// TwinCAT 3 PLC project PlcCode
// ProgramVersion: 3.1.4024.12
// libraries:
//   Tc2_Standard, * (Beckhoff Automation GmbH)
//   Tc2_System, * (Beckhoff Automation GmbH)
//   Tc2_Utilities, * (Beckhoff Automation GmbH)
//   Tc3_IotBase, * (Beckhoff Automation GmbH)
//   Tc3_JsonXml, * (Beckhoff Automation GmbH)
//   Tc3_Module, * (Beckhoff Automation GmbH)
// project tree:
//   GVLs/ GVL.TcGVL
//   / PlcTask.TcTTO
//   POUs/ MAIN.TcPOU
//   ReadConfigFile/CELLS_INFO_STRUCTURES/Development/ DUT_STRUCT_C000000_DEV.TcDUT (not stored), DUT_STRUCT_C000001_DEV.TcDUT (not stored), DUT_STRUCT_C000002_DEV.TcDUT, DUT_STRUCT_C000003_DEV.TcDUT (not stored), DUT_STRUCT_C000004_DEV.TcDUT (not stored), DUT_STRUCT_C000005_DEV.TcDUT, DUT_STRUCT_C000006_DEV.TcDUT (not stored), DUT_STRUCT_C000007_DEV.TcDUT (not stored), DUT_STRUCT_C000008_DEV.TcDUT, DUT_STRUCT_C000009_DEV.TcDUT (not stored), DUT_STRUCT_C000010_DEV.TcDUT (not stored), DUT_STRUCT_C000012_DEV.TcDUT, DUT_STRUCT_LINECONTROLLER_DEV.TcDUT, DUT_STRUCT_TRACKSERVER_DEV.TcDUT
//   ReadConfigFile/CELLS_INFO_STRUCTURES/Production/ DUT_STRUCT_C000000_PROD.TcDUT, DUT_STRUCT_C000001_PROD.TcDUT (not stored), DUT_STRUCT_C000002_PROD.TcDUT, DUT_STRUCT_C000003_PROD.TcDUT (not stored), DUT_STRUCT_C000004_PROD.TcDUT, DUT_STRUCT_C000005_PROD.TcDUT (not stored), DUT_STRUCT_C000006_PROD.TcDUT, DUT_STRUCT_C000007_PROD.TcDUT (not stored), DUT_STRUCT_C000008_PROD.TcDUT (not stored), DUT_STRUCT_C000009_PROD.TcDUT, DUT_STRUCT_C000010_PROD.TcDUT (not stored), DUT_STRUCT_C000012_PROD.TcDUT (not stored), DUT_STRUCT_LINECONTROLLER_PROD.TcDUT, DUT_STRUCT_TRACKSERVER_PROD.TcDUT
//   ReadConfigFile/ DUT_STRUCT_VARIABLES.TcDUT, FB_HttpGet.TcPOU, FB_ReadFile.TcPOU, ST_ReceivedData.TcDUT (not stored)
// real-time tasks:
//   TASK PlcTask: cycle T#10ms, priority 20, ADS port 350
//   TASK PlcTask1: cycle T#10ms, priority 21, ADS port 351

CONFIGURATION PlcCode
    RESOURCE PLC ON TwinCAT3
        TASK PlcTask(INTERVAL := T#10ms, PRIORITY := 20);
        PROGRAM MAIN WITH PlcTask : MAIN;
    END_RESOURCE
END_CONFIGURATION

// ---- ReadConfigFile/CELLS_INFO_STRUCTURES/Development/DUT_STRUCT_C000002_DEV.TcDUT
TYPE DUT_STRUCT_C000002_DEV :
STRUCT
	sCellName			:STRING := 'C000002';
	sIpAddress			:STRING := '';
	sAmsNetId			:STRING := '';
	sOpcUaURL			:STRING := 'opc.tcp://:4840';
	sStation1			:STRING := 'S000007';
END_STRUCT
END_TYPE

// ---- ReadConfigFile/CELLS_INFO_STRUCTURES/Development/DUT_STRUCT_C000005_DEV.TcDUT
TYPE DUT_STRUCT_C000005_DEV :
STRUCT
	sCellName			:STRING := 'C000005';
	sIpAddress			:STRING := '';
	sAmsNetId			:STRING := '';
	sOpcUaURL			:STRING := 'opc.tcp://:4840';
	sStation1			:STRING := 'S000001';
END_STRUCT
END_TYPE

// ---- ReadConfigFile/CELLS_INFO_STRUCTURES/Development/DUT_STRUCT_C000008_DEV.TcDUT
TYPE DUT_STRUCT_C000008_DEV :
STRUCT
	sCellName			:STRING := 'C000008';
	sIpAddress			:STRING := '';
	sAmsNetId			:STRING := '';
	sOpcUaURL			:STRING := 'opc.tcp://:4840';
	sStation1			:STRING := 'S000005';
END_STRUCT
END_TYPE

// ---- ReadConfigFile/CELLS_INFO_STRUCTURES/Development/DUT_STRUCT_C000012_DEV.TcDUT
TYPE DUT_STRUCT_C000012_DEV :
STRUCT
	sCellName			:STRING := 'C000012';
	sIpAddress			:STRING := '';
	sAmsNetId			:STRING := '';
	sOpcUaURL			:STRING := 'opc.tcp://:4840';
	sStation1			:STRING := 'S000010';
END_STRUCT
END_TYPE

// ---- ReadConfigFile/CELLS_INFO_STRUCTURES/Development/DUT_STRUCT_LINECONTROLLER_DEV.TcDUT
TYPE DUT_STRUCT_LINECONTROLLER_DEV :
STRUCT
	sCellName			:STRING := 'LINECONTROLLER';
	sIpAddress			:STRING := '10.155.180.8';
	sAmsNetId			:STRING := '';
END_STRUCT
END_TYPE

// ---- ReadConfigFile/CELLS_INFO_STRUCTURES/Development/DUT_STRUCT_TRACKSERVER_DEV.TcDUT
TYPE DUT_STRUCT_TRACKSERVER_DEV :
STRUCT
	sCellName			:STRING := 'TRACKSERVER';
	sIpAddress			:STRING := '10.155.180.10';
	sAmsNetId			:STRING := '10.155.180.10.1.1';
END_STRUCT
END_TYPE

// ---- ReadConfigFile/CELLS_INFO_STRUCTURES/Production/DUT_STRUCT_C000000_PROD.TcDUT
TYPE DUT_STRUCT_C000000_PROD :
STRUCT
	sCellName			:STRING := 'C000000';
	sIpAddress			:STRING := '10.38.190.130';
	sAmsNetId			:STRING := '10.38.190.130.1.1';
	sOpcUaURL			:STRING := 'opc.tcp://10.38.190.130:4840';
	sUhfRfidOpcUaURL	:STRING := 'opc.tcp://10.38.190.132:4840';
	sHfRfidOpcUaURL		:STRING := 'opc.tcp://10.38.190.134:4840';
	sStation1			:STRING := 'S00000A';
END_STRUCT
END_TYPE

// ---- ReadConfigFile/CELLS_INFO_STRUCTURES/Production/DUT_STRUCT_C000002_PROD.TcDUT
TYPE DUT_STRUCT_C000002_PROD :
STRUCT
	sCellName			:STRING := 'C000002';
	sIpAddress			:STRING := '10.38.191.20';
	sAmsNetId			:STRING := '10.38.191.20.1.1';
	sOpcUaURL			:STRING := 'opc.tcp://10.38.191.20:4840';
	sStation1			:STRING := 'S000007';
END_STRUCT
END_TYPE

// ---- ReadConfigFile/CELLS_INFO_STRUCTURES/Production/DUT_STRUCT_C000004_PROD.TcDUT
TYPE DUT_STRUCT_C000004_PROD :
STRUCT
	sCellName			:STRING := 'C000004';
	sIpAddress			:STRING := '10.38.190.201';
	sAmsNetId			:STRING := '10.38.190.201.1.1';
	sOpcUaURL			:STRING := 'opc.tcp://10.38.190.201:4840';
	sStation1			:STRING := 'S000003';
END_STRUCT
END_TYPE

// ---- ReadConfigFile/CELLS_INFO_STRUCTURES/Production/DUT_STRUCT_C000006_PROD.TcDUT
TYPE DUT_STRUCT_C000006_PROD :
STRUCT
	sCellName			:STRING := 'C000006';
	sIpAddress			:STRING := '10.38.190.200';
	sAmsNetId			:STRING := '10.38.190.200.1.1';
	sOpcUaURL			:STRING := 'opc.tcp://10.38.190.200:4840';
	sStation1			:STRING := 'S000002';
END_STRUCT
END_TYPE

// ---- ReadConfigFile/CELLS_INFO_STRUCTURES/Production/DUT_STRUCT_C000009_PROD.TcDUT
TYPE DUT_STRUCT_C000009_PROD :
STRUCT
	sCellName			:STRING := 'C000009';
	sIpAddress			:STRING := '10.38.191.60';
	sAmsNetId			:STRING := '10.38.191.60.1.1';
	sOpcUaURL			:STRING := 'opc.tcp://10.38.191.60:4840';
	sUhfRfidOpcUaURL	:STRING := 'opc.tcp://10.38.190.132:4840';
	sHfRfidOpcUaURL		:STRING := 'opc.tcp://10.38.191.66:4840';
	sStation1			:STRING := 'S000004';
	sLastingPC			:STRING := '10.38.191.65';
END_STRUCT
END_TYPE

// ---- ReadConfigFile/CELLS_INFO_STRUCTURES/Production/DUT_STRUCT_LINECONTROLLER_PROD.TcDUT
TYPE DUT_STRUCT_LINECONTROLLER_PROD :
STRUCT
	sCellName			:STRING := 'LINECONTROLLER';
	sIpAddress			:STRING := '10.38.190.120';
	sAmsNetId			:STRING := '';
END_STRUCT
END_TYPE

// ---- ReadConfigFile/CELLS_INFO_STRUCTURES/Production/DUT_STRUCT_TRACKSERVER_PROD.TcDUT
TYPE DUT_STRUCT_TRACKSERVER_PROD :
STRUCT
	sCellName			:STRING := 'TRACKSERVER';
	sIpAddress			:STRING := '10.38.190.121';
	sAmsNetId			:STRING := '10.38.190.121.1.1';
END_STRUCT
END_TYPE

// ---- ReadConfigFile/DUT_STRUCT_VARIABLES.TcDUT
TYPE DUT_STRUCT_VARIABLES :
STRUCT
	sCellName			:STRING;
	sIpAddress			:STRING;
	sAmsNetId			:STRING;
	sOpcUaURL			:STRING;
	sUhfRfidOpcUaURL	:STRING;
	sHfRfidOpcUaURL		:STRING;
	sStation1			:STRING;
	sStation2			:STRING;
END_STRUCT
END_TYPE

// ---- GVLs/GVL.TcGVL
{attribute 'qualified_only'}
VAR_GLOBAL
	
	// vars for JSON & HTTP GET response
	sString						:ARRAY[0..100] OF STRING(255);
	jsonFileResult 				:STRING(501);

	// repo info
	sRelease					:STRING;
	sCommitID					:STRING;
	sTag						:STRING;
	
	// cells info
	C000000						:DUT_STRUCT_VARIABLES;
	C000001						:DUT_STRUCT_VARIABLES;
	C000002						:DUT_STRUCT_VARIABLES;
	C000003						:DUT_STRUCT_VARIABLES;
	C000004						:DUT_STRUCT_VARIABLES;
	C000005						:DUT_STRUCT_VARIABLES;
	C000006						:DUT_STRUCT_VARIABLES;
	C000007						:DUT_STRUCT_VARIABLES;
	C000008						:DUT_STRUCT_VARIABLES;
	C000009						:DUT_STRUCT_VARIABLES;
	C000010						:DUT_STRUCT_VARIABLES;
	C000012						:DUT_STRUCT_VARIABLES;
	LineController				:DUT_STRUCT_VARIABLES;
	Trackserver					:DUT_STRUCT_VARIABLES;
	
	// cells info for PRODUCTION
//	C000000_PROD				:DUT_STRUCT_C000000_PROD;
//	C000001_PROD				:DUT_STRUCT_C000001_PROD;
//	C000002_PROD				:DUT_STRUCT_C000002_PROD;
//	C000003_PROD				:DUT_STRUCT_C000003_PROD;
//	C000004_PROD				:DUT_STRUCT_C000004_PROD;
//	C000005_PROD				:DUT_STRUCT_C000005_PROD;
//	C000006_PROD				:DUT_STRUCT_C000006_PROD;
//	C000007_PROD				:DUT_STRUCT_C000007_PROD;
//	C000008_PROD				:DUT_STRUCT_C000008_PROD;
//	C000009_PROD				:DUT_STRUCT_C000009_PROD;
//	C000010_PROD				:DUT_STRUCT_C000010_PROD;
//	C000012_PROD				:DUT_STRUCT_C000012_PROD;
//	TrackServer_PROD			:DUT_STRUCT_TRACKSERVER_PROD;
//	LineController_PROD			:DUT_STRUCT_LINECONTROLLER_PROD;
	
//	// cells info for DEVELOPMENT
//	C000000_DEV					:DUT_STRUCT_C000000_DEV;
//	C000001_DEV					:DUT_STRUCT_C000001_DEV;
//	C000002_DEV					:DUT_STRUCT_C000002_DEV;
//	C000003_DEV					:DUT_STRUCT_C000003_DEV;
//	C000004_DEV					:DUT_STRUCT_C000004_DEV;
//	C000005_DEV					:DUT_STRUCT_C000005_DEV;
//	C000006_DEV					:DUT_STRUCT_C000006_DEV;
//	C000007_DEV					:DUT_STRUCT_C000007_DEV;
//	C000008_DEV					:DUT_STRUCT_C000008_DEV;
//	C000009_DEV					:DUT_STRUCT_C000009_DEV;
//	C000010_DEV					:DUT_STRUCT_C000010_DEV;
//	C000012_DEV					:DUT_STRUCT_C000012_DEV;
//	TrackServer_DEV				:DUT_STRUCT_TRACKSERVER_DEV;
//	LineController_DEV			:DUT_STRUCT_LINECONTROLLER_DEV;
END_VAR

// ---- POUs/MAIN.TcPOU
PROGRAM MAIN

VAR
	// develop branch
	fbReadFile					:FB_ReadFile;
	bHttpGet					:BOOL := TRUE;

    fbHttpClient				:FB_IotHttpClient := (sHostName:='api.github.com', bKeepAlive:=TRUE, tConnectionTimeout:=T#10S);
    fbHttpGetOpen				:FB_HttpGet;
END_VAR

fbReadFile();

// HTTP GET request
IF NOT fbHttpClient.bConfigured THEN
    fbHttpClient.nHostPort := 443;
    fbHttpClient.stTLS.bNoServerCertCheck := TRUE;
END_IF

IF fbHttpClient.bConfigured THEN
    fbHttpGetOpen(bSend := bHttpGet, fbClient := fbHttpClient);
END_IF

fbHttpClient.Execute();

END_PROGRAM

// ---- ReadConfigFile/FB_ReadFile.TcPOU
FUNCTION_BLOCK FB_ReadFile

VAR
	CSVMemBufferReader		:FB_CSVMemBufferReader;
	fbFileOpen				:FB_FileOpen;
	fbFileGet				:FB_FileGets;
	fbFileClose				:FB_FileClose;
	
	sPathName				:STRING := 'C:\RUO folder\Configuration file branches TEST\';
	sFileName				:STRING := '\test-branches-config-file\PROD_MasterConfig.txt';
	sConfigPathFile			:STRING(300) := CONCAT(sPathName, sFileName);
	
	bReset					:BOOL;
	nCol					:INT;
	hFile					:UINT;
	value					:STRING[300];
	sBufferString			:ARRAY[0..100]OF STRING;
	iStep					:INT;
	sLine					:STRING;
	nRow					:INT;
	bRead					:BOOL := true;
	bEOF					:BOOL;
	i						:INT;
	iCRLFCounter			:INT;
	
	// split string
	aSplit					:ARRAY[0..cMax] OF STRING(255);
	bResultSplit			:BOOL;
	ii						:UDINT;
END_VAR
VAR CONSTANT
	cStepInit				:INT := 0;
	cStepOpenFile			:INT := 10;
	cStepGetLine			:INT := 20;
	cStepEOFCheck			:INT := 25;
	cStepReadLine			:INT := 30;
	cStepParseData			:INT := 35;
	cStepCloseFile			:INT := 40;
	cStepError				:INT := 8000;
	
	// split string
	cMax					:UDINT := 100;
END_VAR

CASE iStep OF
	
	cStepInit:
	
		//* semicolon (;) := 16#3B => german field separator, comma (,) := 16#2C => US field separator
		DEFAULT_CSV_FIELD_SEP := 16#3B;
		
		nRow := 0;
		nCol := 0;
		iCRLFCounter := 0;
		bEOF := FALSE;
		bReset := FALSE;
		
		// fb Reset
		fbFileOpen(bExecute := FALSE);
		fbFileClose(bExecute := FALSE);
		fbFileGet(bExecute := FALSE);
			
		IF bRead 
			AND NOT fbfileopen.bBusy
			AND NOT fbfileclose.bBusy
			AND NOT fbfileget.bBusy
			THEN
			
			FOR i := 0 TO 24 DO
				GVL.sString[i] := '';
				
			END_FOR
			iStep := cStepOpenFile;
			bRead := FALSE;
		END_IF;
		
		cStepOpenFile:
			fbFileopen(	sNetId := '', sPathName := sConfigPathFile, nMode := FOPEN_MODEREAD,
						ttimeout := T#3S, ePath := E_OpenPath.PATH_GENERIC, bExecute := TRUE, hFile => hfile);
					
		IF NOT fbfileopen.bBusy THEN
			IF fbfileopen.bError THEN
				iStep := cStepError;	
			ELSE
				iStep := cStepGetLine;
			END_IF
		END_IF
		
		cStepGetLine:
			fbFileGet(hFile := hFile, bExecute := TRUE, sLine => sLine);
	
		IF NOT fbFileGet.bBusy THEN
			IF fbFileGet.bError THEN
				iStep := cStepError;	
			ELSE IF fbFileGet.bEOF THEN
				bEOF := TRUE;
			END_IF
		(*
			IF RIGHT( Fileget.sLine, 1 ) = '$N' THEN
				sCSVLine := REPLACE( sCSVLine, '$R$L', 2, LEN( sCSVLine ) );
			END_IF
		*)
			iStep := cStepEOFCheck;
			END_IF
		END_IF
		
		cStepEOFCheck:
				fbFileGet(bExecute := FALSE);
		IF bEOF THEN
			iStep := cStepCloseFile;
		ELSE
			iStep := cStepReadLine;	
		END_IF
	
		cStepReadLine:
			nCol := 0;
			CSVMemBufferReader.eCmd := E_EnumCmdType.eEnumCmd_First;
				REPEAT
					CSVMemBufferReader(pBuffer := ADR(sLine), cbBuffer := SIZEOF(sLine), getValue => value);
				
					IF CSVMemBufferReader.bOk THEN
						sBufferString[ncol] := value;
						CSVMemBufferReader.eCmd := E_EnumCmdType.eEnumCmd_Next;
						ncol := ncol + 1;
						IF CSVMemBufferReader.bCRLF THEN
							iCRLFCounter := iCRLFCounter + 1;
						END_IF
					END_IF
				UNTIL NOT CSVMemBufferReader.bOk 
				END_REPEAT	
			istep := cStepParseData;
			
		cStepParseData:
			// check EOF
			IF fbFileGet.bEOF THEN
				iStep := cStepCloseFile;
			ELSE
				GVL.sString[nRow] := sBufferString[0];
				nRow := nRow + 1;
				iStep := cStepGetLine;
			END_IF
		
		cStepCloseFile:	
			fbFileClose(hFile := hFile, bExecute := TRUE);
			IF NOT fbFileClose.bBusy THEN
				IF fbFileClose.bError THEN
					iStep := cStepError;	
				END_IF
			ELSE
				fbFileClose(bExecute:=FALSE);
				iStep := cStepInit;
			END_IF
			
		cStepError:
			IF bReset THEN
				iStep := cStepInit;
			END_IF
END_CASE

// split/parse strings
FOR ii := 0 TO cMax - 1 DO
	
	aSplit[ii] := GVL.sString[ii];
	bResultSplit := FindAndSplitChar(sSeparatorChar := '=', pSrcString := ADR(aSplit[ii]),
									  pLeftString := ADR(aSplit[ii + 1]), nLeftSize := SIZEOF(aSplit[ii + 1]),
									  pRightString := ADR(aSplit[ii]), nRightSize := SIZEOF(aSplit[ii]),
									  bSearchFromRight := FALSE);
									  
	// assign values from config file
	// cell 00
	GVL.C000000.sCellName 			:= aSplit[0];
	GVL.C000000.sIpAddress 			:= aSplit[1];
	GVL.C000000.sAmsNetId 			:= aSplit[2];
	GVL.C000000.sOpcUaURL 			:= aSplit[3];
	GVL.C000000.sUhfRfidOpcUaURL 	:= aSplit[4];
	GVL.C000000.sHfRfidOpcUaURL		:= aSplit[5];
	GVL.C000000.sStation1		 	:= aSplit[6];
	
	// cell 01
	GVL.C000001.sCellName 			:= aSplit[7];
	GVL.C000001.sIpAddress 			:= aSplit[8];
	GVL.C000001.sAmsNetId 			:= aSplit[9];
	GVL.C000001.sOpcUaURL 			:= aSplit[10];
	GVL.C000001.sStation1		 	:= aSplit[11];
	GVL.C000001.sStation2		 	:= aSplit[12];
	
	// cell 02
	GVL.C000002.sCellName 			:= aSplit[13];
	GVL.C000002.sIpAddress 			:= aSplit[14];
	GVL.C000002.sAmsNetId 			:= aSplit[15];
	GVL.C000002.sOpcUaURL 			:= aSplit[16];
	GVL.C000002.sStation1		 	:= aSplit[17];
	
	// cell 03
	GVL.C000003.sCellName 			:= aSplit[18];
	GVL.C000003.sIpAddress 			:= aSplit[19];
	GVL.C000003.sAmsNetId 			:= aSplit[20];
	GVL.C000003.sOpcUaURL 			:= aSplit[21];
	GVL.C000003.sStation1		 	:= aSplit[22];
	
	// cell 04
	GVL.C000004.sCellName 			:= aSplit[23];
	GVL.C000004.sIpAddress 			:= aSplit[24];
	GVL.C000004.sAmsNetId 			:= aSplit[25];
	GVL.C000004.sOpcUaURL 			:= aSplit[26];
	GVL.C000004.sStation1		 	:= aSplit[27];
	
	// cell 05
	GVL.C000005.sCellName 			:= aSplit[28];
	GVL.C000005.sIpAddress 			:= aSplit[29];
	GVL.C000005.sAmsNetId 			:= aSplit[30];
	GVL.C000005.sOpcUaURL 			:= aSplit[31];
	GVL.C000005.sStation1		 	:= aSplit[32];
	
	// cell 06
	GVL.C000006.sCellName 			:= aSplit[33];
	GVL.C000006.sIpAddress 			:= aSplit[34];
	GVL.C000006.sAmsNetId 			:= aSplit[35];
	GVL.C000006.sOpcUaURL 			:= aSplit[36];
	GVL.C000006.sStation1		 	:= aSplit[37];
	
	// cell 07
	GVL.C000007.sCellName 			:= aSplit[38];
	GVL.C000007.sIpAddress 			:= aSplit[39];
	GVL.C000007.sAmsNetId 			:= aSplit[40];
	GVL.C000007.sOpcUaURL 			:= aSplit[41];
	GVL.C000007.sStation1		 	:= aSplit[42];
	
	// cell 08
	GVL.C000008.sCellName 			:= aSplit[43];
	GVL.C000008.sIpAddress 			:= aSplit[44];
	GVL.C000008.sAmsNetId 			:= aSplit[45];
	GVL.C000008.sOpcUaURL 			:= aSplit[46];
	GVL.C000008.sStation1		 	:= aSplit[47];
	
	// cell 09
	GVL.C000009.sCellName 			:= aSplit[48];
	GVL.C000009.sIpAddress 			:= aSplit[49];
	GVL.C000009.sAmsNetId 			:= aSplit[50];
	GVL.C000009.sOpcUaURL 			:= aSplit[51];
	GVL.C000009.sUhfRfidOpcUaURL 	:= aSplit[52];
	GVL.C000009.sHfRfidOpcUaURL		:= aSplit[53];
	GVL.C000009.sStation1		 	:= aSplit[54];
	
	// cell 10
	GVL.C000010.sCellName 			:= aSplit[55];
	GVL.C000010.sIpAddress 			:= aSplit[56];
	GVL.C000010.sAmsNetId 			:= aSplit[57];
	GVL.C000010.sOpcUaURL 			:= aSplit[58];
	GVL.C000010.sStation1		 	:= aSplit[59];
	GVL.C000010.sStation2		 	:= aSplit[60];
	
	// cell 12
	GVL.C000012.sCellName 			:= aSplit[61];
	GVL.C000012.sIpAddress 			:= aSplit[62];
	GVL.C000012.sAmsNetId 			:= aSplit[63];
	GVL.C000012.sOpcUaURL		 	:= aSplit[64];
	GVL.C000012.sStation1		 	:= aSplit[65];
	
	// linecontroller
	GVL.LineController.sCellName 	:= aSplit[66];
	GVL.LineController.sIpAddress 	:= aSplit[67];
	GVL.LineController.sAmsNetId 	:= aSplit[68];
	
	// trackserver
	GVL.Trackserver.sCellName 		:= aSplit[69];
	GVL.Trackserver.sIpAddress 		:= aSplit[70];
	GVL.Trackserver.sAmsNetId 		:= aSplit[71];
	
	IF NOT bResultSplit THEN
		EXIT;
	END_IF
END_FOR

END_FUNCTION_BLOCK

// ---- ReadConfigFile/FB_HttpGet.TcPOU
FUNCTION_BLOCK FB_HttpGet

VAR_INPUT
    bSend				:BOOL;
END_VAR

VAR_IN_OUT
    fbClient			:FB_IotHttpClient;
END_VAR

VAR_OUTPUT
    bBusy				:BOOL;
    bError				:BOOL;
END_VAR

VAR
    fbRequest			:FB_IotHttpRequest;
    fbJson				:FB_JsonDomParser;
    nState				:UDINT;
    RisingEdge			:R_TRIG;

    bGetContentResult 	:BOOL;
    sContent			:STRING(511);

    bGetJsonResult		:BOOL;
    jsonDoc				:SJsonValue;
    jsonVal				:SJsonValue;
    sResultValue      	:STRING;

    nReqCount			:UDINT;
    nResCount			:UDINT;
    nValidResCount		:UDINT;
    nErrCount			:UDINT;
	
	// split string
	aSplit				:ARRAY[0..cMax] OF STRING(501);
	aLeftSplit			:ARRAY[1..cMax] OF STRING(501);
	aRightSplit			:ARRAY[1..cMax] OF STRING(501);
	bResultSplit		:BOOL;
	ii					:UDINT;
	
	// JSON parse
	jsonProp			:SJsonValue;
	jsonValue			:SJsonValue;
	bHasMember			:BOOL;
	stReceivedData		:ST_ReceivedData;
END_VAR
VAR CONSTANT
	cMax				:UDINT := 15;
END_VAR

RisingEdge(CLK := bSend);
CASE nState OF
0:
    IF RisingEdge.Q THEN
        IF fbRequest.SendRequest(sUri := '/repos/ECCO-RUO/test-branches-config-file/tags',
                                 fbClient := fbClient, 
                                 eRequestType := ETcIotHttpRequestType.HTTP_Get, 0, 0, 0) THEN
            nState := 1;
            nReqCount := nReqCount+1;
            bBusy := TRUE;
            bError := FALSE;
        END_IF
    END_IF
1:
    IF NOT fbRequest.bBusy THEN
        bError := TRUE;
        IF NOT fbRequest.bError THEN
            bGetContentResult := fbRequest.GetContent(pContent := ADR(sContent), 
                                                     nContentSize := SIZEOF(sContent), 
                                                     bSetNullTermination := TRUE);
            IF fbRequest.nStatusCode >= 200 AND fbRequest.nStatusCode < 300 THEN
                bGetJsonResult := FALSE;
                jsonDoc := fbRequest.GetJsonDomContent(fbJson);
                IF jsonDoc <> 0 THEN
					nValidResCount := nValidResCount+1;
                    bError := FALSE;
                END_IF
                nResCount := nResCount+1;
            END_IF
        END_IF
        nState := 0;
        bBusy := FALSE;
        IF bError THEN
            nErrCount := nErrCount+1;
        END_IF
    END_IF
END_CASE

// split JSON HTTP GET response from REPO
aLeftSplit[1] := sContent;
FOR ii := 1 TO cMax-1 DO					  
	bResultSplit := FindAndSplitChar(sSeparatorChar := '[', pSrcString := ADR(aLeftSplit[ii]),
									  pLeftString := ADR(aLeftSplit[ii + 1]), nLeftSize := SIZEOF(aLeftSplit[ii + 1]),
									  pRightString := ADR(aLeftSplit[ii]), nRightSize := SIZEOF(aLeftSplit[ii]),
									  bSearchFromRight := FALSE);  
 
	bResultSplit := FindAndSplitChar(sSeparatorChar := ']', pSrcString := ADR(aLeftSplit[ii]),
									  pLeftString := ADR(aRightSplit[ii + 1]), nLeftSize := SIZEOF(aRightSplit[ii + 1]),
									  pRightString := ADR(aRightSplit[ii]), nRightSize := SIZEOF(aRightSplit[ii]),
									  bSearchFromRight := FALSE);
GVL.jsonFileResult := aRightSplit[2];
								  
    IF NOT bResultSplit THEN
        EXIT;
    END_IF
END_FOR
					
// get TAG from REPO
jsonDoc := fbJson.ParseDocument(GVL.jsonFileResult);
bHasMember := fbJson.HasMember(jsonDoc, 'name');
IF (bHasMember) THEN
  bHasMember := FALSE;
  jsonProp := fbJson.FindMember(jsonDoc, 'name');
  stReceivedData.name := fbJson.GetString(jsonProp);
END_IF

bHasMember := fbJson.HasMember(jsonDoc, 'tarball_url');
IF (bHasMember) THEN
  bHasMember := FALSE;
  jsonProp := fbJson.FindMember(jsonDoc, 'tarball_url');
  stReceivedData.tarball_url := fbJson.GetString(jsonProp);
END_IF

bHasMember := fbJson.HasMember(jsonDoc, 'zipball_url');
IF (bHasMember) THEN
  bHasMember := FALSE;
  jsonProp := fbJson.FindMember(jsonDoc, 'zipball_url');
  stReceivedData.zipball_url := fbJson.GetString(jsonProp);
END_IF

GVL.sTag := stReceivedData.name;
GVL.sCommitID := stReceivedData.tarball_url;
GVL.sRelease := stReceivedData.zipball_url;

END_FUNCTION_BLOCK
